FUNCTION_BLOCK InjectorPumpsController
  (* Standard: 61499-2 *)
  (* Version 0.1, 2016-00-28, hpea485, UOA *)
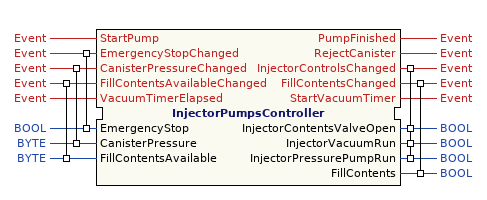
  EVENT_INPUT
    StartPump;
    EmergencyStopChanged WITH EmergencyStop;
    CanisterPressureChanged WITH CanisterPressure;
    FillContentsAvailableChanged WITH FillContentsAvailable;
    VacuumTimerElapsed;
  END_EVENT
  EVENT_OUTPUT
    PumpFinished;
    RejectCanister;
    InjectorControlsChanged WITH InjectorPressurePumpRun, InjectorVacuumRun, InjectorContentsValveOpen;
    FillContentsChanged WITH FillContents;
    StartVacuumTimer;
  END_EVENT
  VAR_INPUT
    EmergencyStop : BOOL;
    CanisterPressure : BYTE;
    FillContentsAvailable : BYTE;
  END_VAR
  VAR_OUTPUT
    InjectorContentsValveOpen : BOOL;
    InjectorVacuumRun : BOOL;
    InjectorPressurePumpRun : BOOL;
    FillContents : BOOL;
  END_VAR
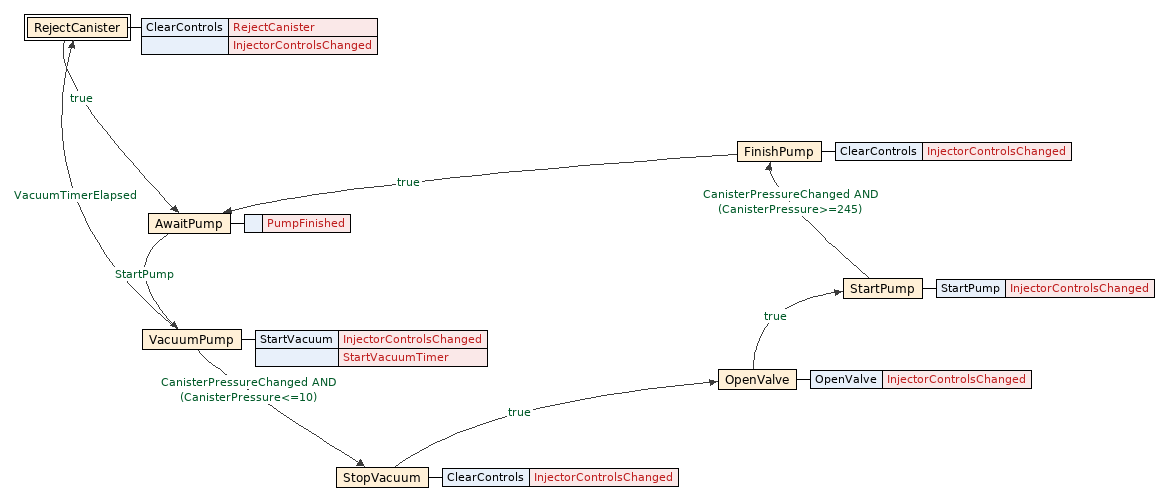
  EC_STATES
    RejectCanister : ClearControls -> RejectCanister, -> InjectorControlsChanged;
    AwaitPump : -> PumpFinished;
    VacuumPump : StartVacuum -> InjectorControlsChanged, -> StartVacuumTimer;
    FinishPump : ClearControls -> InjectorControlsChanged;
    StartPump : StartPump -> InjectorControlsChanged;
    OpenValve : OpenValve -> InjectorControlsChanged;
    StopVacuum : ClearControls -> InjectorControlsChanged;
  END_STATES
  EC_TRANSITIONS
    RejectCanister TO AwaitPump := true;
    AwaitPump TO VacuumPump := StartPump;
    VacuumPump TO RejectCanister := VacuumTimerElapsed;
    VacuumPump TO StopVacuum := CanisterPressureChanged AND (CanisterPressure<=10);
    FinishPump TO AwaitPump := true;
    StartPump TO FinishPump := CanisterPressureChanged AND (CanisterPressure>=245);
    OpenValve TO StartPump := true;
    StopVacuum TO OpenValve := true;
  END_TRANSITIONS
  ALGORITHM StartVacuum IN VHDL:
me->InjectorVacuumRun = 1;
//printf("Injector: Start vacuum\n");
  END_ALGORITHM
  ALGORITHM ClearControls IN VHDL:
me->InjectorContentsValveOpen = 0;
me->InjectorPressurePumpRun = 0;
me->InjectorVacuumRun = 0;
//printf("Injector: Clear controls\n");
  END_ALGORITHM
  ALGORITHM OpenValve IN VHDL:
me->InjectorContentsValveOpen = 1;
//printf("Injector: Open valve\n");
  END_ALGORITHM
  ALGORITHM StartPump IN VHDL:
me->InjectorPressurePumpRun = 1;
//printf("Injector: Start pump\n");
  END_ALGORITHM
END_FUNCTION_BLOCK
